{attribute 'qualified_only'}
{attribute 'strict'}
{attribute 'to_string'}
TYPE E_WaferTransferCmd :
(
	None := 0,
	PrepareSend,
	PrepareReceive,
	SendMaterial,
	ReceiveMaterial
);
END_TYPE

(* stored: Version 1.1.0.1, ProductVersion 3.1.4026.18
   DUT E_WaferTransferCmd: Id {4710c465-4442-47c0-8c1d-fa9ad0dfeca8} *)
